(* LS Electric XG5000 project: 241004_실습4램프작동_내부변수사용 *)
(* PLC LSPLC *)

PROGRAM NewProgram (* task: 스캔 프로그램 *)
VAR
    내부변수 AT %MX3 : BOOL;
    녹색램프 AT %MX0 : BOOL;
    램프1 AT %QX0.1.0 : BOOL;
    램프2 AT %QX0.1.1 : BOOL;
    램프3 AT %QX0.1.2 : BOOL;
    버튼1 AT %IX0.0.0 : BOOL;
    버튼2 AT %IX0.0.1 : BOOL;
    적색램프 AT %MX2 : BOOL;
    황색램프 AT %MX1 : BOOL;
END_VAR
VAR
    _e1 : R_TRIG;
    _e2 : R_TRIG;
END_VAR

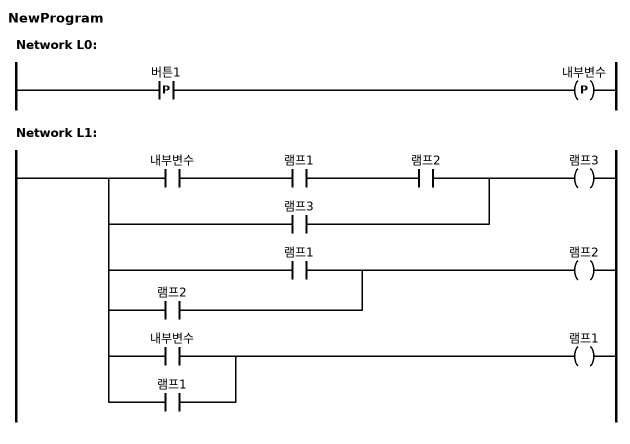
(* Rung L0 *)
_e1(CLK := 버튼1);
_e2(CLK := _e1.Q);
내부변수 := _e2.Q;
(* Rung L1 *)
램프3 := (내부변수 AND 램프1 AND 램프2) OR 램프3;
램프2 := 램프1 OR 램프2;
램프1 := 내부변수 OR 램프1;
END_PROGRAM